(* Logix 5000 project; controller KTC_lab3 vendor 1 type 14 code 150 rev 30.11; software revision 30.00 *)

TASK MainTask (continuous, watchdog 500 ms) : MainProgram

MODULES
   Local : vendor 1 type 14 code 150 (Compact 0, rev 30.11)
      Counters : Embedded (Compact 3, rev 1.1, Output RPI 20 ms)
      Discrete_IO : Embedded (Compact 1, rev 3.1, Output RPI 20 ms)
      Analog_IO : Embedded (Compact 2, rev 1.1, Output RPI 80 ms)
END_MODULES

PROGRAM MainProgram   (* main routine MainRoutine *)
VAR
   PB0 : ALIAS FOR Local:1:I.Data.0;   // PBNO
   PB2 : ALIAS FOR Local:1:I.Data.2;   // PBNC2
   PL1 : ALIAS FOR Local:1:O.Data.1;   // LIGHT 1
END_VAR

ROUTINE MainRoutine   (* ladder *)
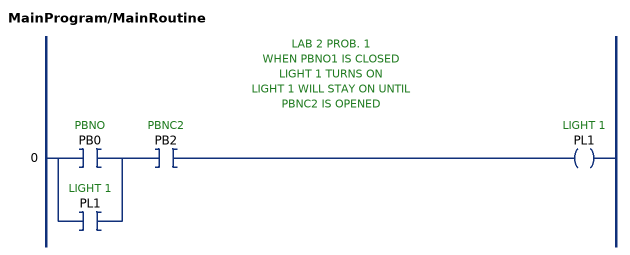
   // LAB 2 PROB. 1
   // WHEN PBNO1 IS CLOSED
   // LIGHT 1 TURNS ON
   // LIGHT 1 WILL STAY ON UNTIL
   // PBNC2 IS OPENED
   0: [XIC(PB0) ,XIC(PL1) ]XIC(PB2)OTE(PL1);
END_ROUTINE
END_PROGRAM
